INTERFACE I_TcUnitRunner

METHOD RunFunctionBlocksTests
END_METHOD

END_INTERFACE

(* stored: Version 1.1.0.1, ProductVersion 3.1.4022.12
   Itf I_TcUnitRunner: Id {ee464aaf-65d4-40d9-bd96-c7f35154f639}
   Method RunFunctionBlocksTests: Id {553a8982-7df2-4993-817e-99230c9d6489} *)
